FUNCTION_BLOCK TMS_Mover EXTENDS FB_Mover
VAR_INPUT
	XtsTrack : IXtsTrack;
	StateMachine : IPmlStateMachine;
END_VAR
VAR_OUTPUT
END_VAR
VAR
	mcActivateTrack : Tc3_McCollisionAvoidance.MC_ActivateTrack;
	mcReadTrackPositions : Tc3_McCollisionAvoidance.MC_ReadTrackPositions;
	MoverActiveTrack : OTCID;
	moverSequence : TmsMoverSequence;
END_VAR
VAR_IN_OUT
	StationArray : ARRAY[*] OF IProcess;
END_VAR

SUPER^();
IF _identInGroup <> 0 THEN
	mcReadTrackPositions(
		Axis:= THIS^._axis, 
		Enable:= TRUE, 
		Valid=> , 
		Busy=> , 
		TrackPosition=> , 
		TrackId=> , 
		PartPosition=> , 
		PartId=> , 
		Error=> , 
		ErrorId=> );
END_IF
mcActivateTrack(Axis := THIS^._axis);
moverSequence(ThisMover := THIS^,
				XtsTrack := XtsTrack,
				StateMachine := StateMachine);

METHOD ActivateTrack : BOOL
VAR_INPUT
	newTrack : OTCID;
END_VAR
IF NOT mcActivateTrack.Busy THEN
	mcActivateTrack.Execute := TRUE;
	mcActivateTrack.TrackId := newTrack;
END_IF
END_METHOD

METHOD PUBLIC SetTrackId : BOOL
VAR_INPUT
	
END_VAR
END_METHOD

END_FUNCTION_BLOCK

(* stored: Version 1.1.0.1, ProductVersion 3.1.4024.11
   POU TMS_Mover: Id {6b131325-7dfb-4240-b139-8c4216101462}, SpecialFunc None
   Method ActivateTrack: Id {5f8dc4a4-b7cd-44e5-baab-59a89ea4550d}
   Method SetTrackId: Id {f860ba64-8391-49dd-9256-26b78ef744f7} *)
